LIN {X 0,Y 101.433,Z 824.046,A -85,B 0,C 180,E1 -28794.73,E2 -28794.73} C_VEL
LIN {X 0,Y 101.287,Z 822.969,A -85,B 0,C 180,E1 -28797.017,E2 -28797.017} C_VEL
LIN {X 0,Y 101.21,Z 822.785,A -85,B 0,C 180,E1 -28800.994,E2 -28800.994} C_VEL
LIN {X 0,Y 101.343,Z 823.216,A -85,B 0,C 180,E1 -28803.478,E2 -28803.478} C_VEL
LIN {X 0,Y 102.456,Z 826.592,A -85,B 0,C 180,E1 -28810.373,E2 -28810.373} C_VEL
LIN {X 0,Y 103.056,Z 827.637,A -85,B 0,C 180,E1 -28812.367,E2 -28812.367} C_VEL
LIN {X 0,Y 104.99,Z 831.596,A -85,B 0,C 180,E1 -28817.358,E2 -28817.358} C_VEL
LIN {X 0,Y 106.785,Z 835.312,A -85,B 0,C 180,E1 -28820.877,E2 -28820.877} C_VEL
LIN {X 0,Y 109.032,Z 840.682,A -85,B 0,C 180,E1 -28824.688,E2 -28824.688} C_VEL
LIN {X 0,Y 109.43,Z 842.378,A -85,B 0,C 180,E1 -28825.48,E2 -28825.48} C_VEL
LIN {X 0,Y 107.888,Z 851.485,A -85,B 0,C 180,E1 -28826.117,E2 -28826.117} C_VEL
LIN {X 0,Y 105.588,Z 860.247,A -85,B 0,C 180,E1 -28826.892,E2 -28826.892} C_VEL
LIN {X 0,Y 102.409,Z 869.139,A -85,B 0,C 180,E1 -28827.923,E2 -28827.923} C_VEL
LIN {X 0,Y 98.739,Z 877.424,A -85,B 0,C 180,E1 -28829.317,E2 -28829.317} C_VEL
LIN {X 0,Y 93.703,Z 886.663,A -85,B 0,C 180,E1 -28831.443,E2 -28831.443} C_VEL
LIN {X 0,Y 87.262,Z 896.197,A -85,B 0,C 180,E1 -28834.634,E2 -28834.634} C_VEL
LIN {X 0,Y 82.122,Z 902.568,A -85,B 0,C 180,E1 -28837.663,E2 -28837.663} C_VEL
LIN {X 0,Y 77.037,Z 908.064,A -85,B 0,C 180,E1 -28841.181,E2 -28841.181} C_VEL
LIN {X 0,Y 71.22,Z 913.622,A -85,B 0,C 180,E1 -28846.31,E2 -28846.31} C_VEL
LIN {X 0,Y 65.132,Z 918.794,A -85,B 0,C 180,E1 -28853.596,E2 -28853.596} C_VEL
LIN {X 0,Y 60.395,Z 922.598,A -85,B 0,C 180,E1 -28862.259,E2 -28862.259} C_VEL
LIN {X 0,Y 58.05,Z 924.345,A -85,B 0,C 180,E1 -28868.703,E2 -28868.703} C_VEL
LIN {X 0,Y 56.461,Z 925.598,A -85,B 0,C 180,E1 -28875.585,E2 -28875.585} C_VEL
LIN {X 0,Y 55.612,Z 926.377,A -85,B 0,C 180,E1 -28882.74,E2 -28882.74} C_VEL
LIN {X 0,Y 55.517,Z 926.675,A -85,B 0,C 180,E1 -28890,E2 -28890} C_VEL
LIN {X 0,Y 55.608,Z 926.364,A -85,B 0,C 180,E1 -28897.261,E2 -28897.261} C_VEL
LIN {X 0,Y 56.456,Z 925.559,A -85,B 0,C 180,E1 -28904.417,E2 -28904.417} C_VEL
LIN {X 0,Y 58.05,Z 924.28,A -85,B 0,C 180,E1 -28911.297,E2 -28911.297} C_VEL
LIN {X 0,Y 61.83,Z 921.345,A -85,B 0,C 180,E1 -28920.764,E2 -28920.764} C_VEL
LIN {X 0,Y 65.131,Z 918.672,A -85,B 0,C 180,E1 -28926.404,E2 -28926.404} C_VEL
LIN {X 0,Y 71.219,Z 913.465,A -85,B 0,C 180,E1 -28933.691,E2 -28933.691} C_VEL
LIN {X 0,Y 78.247,Z 906.598,A -85,B 0,C 180,E1 -28939.769,E2 -28939.769} C_VEL
LIN {X 0,Y 84.745,Z 899.107,A -85,B 0,C 180,E1 -28943.958,E2 -28943.958} C_VEL
LIN {X 0,Y 90.162,Z 891.744,A -85,B 0,C 180,E1 -28946.898,E2 -28946.898} C_VEL
LIN {X 0,Y 95.147,Z 883.805,A -85,B 0,C 180,E1 -28949.168,E2 -28949.168} C_VEL
LIN {X 0,Y 100.175,Z 873.929,A -85,B 0,C 180,E1 -28951.279,E2 -28951.279} C_VEL
LIN {X 0,Y 104.464,Z 863.001,A -85,B 0,C 180,E1 -28952.767,E2 -28952.767} C_VEL
LIN {X 0,Y 107.227,Z 853.306,A -85,B 0,C 180,E1 -28953.673,E2 -28953.673} C_VEL
LIN {X 0,Y 109.052,Z 843.744,A -85,B 0,C 180,E1 -28954.304,E2 -28954.304} C_VEL
LIN {X 0,Y 109.146,Z 841.961,A -85,B 0,C 180,E1 -28954.566,E2 -28954.566} C_VEL
LIN {X 0,Y 108.33,Z 839.135,A -85,B 0,C 180,E1 -28956.079,E2 -28956.079} C_VEL
LIN {X 0,Y 105.726,Z 833.29,A -85,B 0,C 180,E1 -28960.588,E2 -28960.588} C_VEL
LIN {X 0,Y 103.976,Z 829.899,A -85,B 0,C 180,E1 -28964.314,E2 -28964.314} C_VEL
LIN {X 0,Y 102.466,Z 826.786,A -85,B 0,C 180,E1 -28968.628,E2 -28968.628} C_VEL
LIN {X 0,Y 101.185,Z 823.736,A -85,B 0,C 180,E1 -28974.895,E2 -28974.895} C_VEL
LIN {X 0,Y 101.064,Z 822.89,A -85,B 0,C 180,E1 -28976.512,E2 -28976.512} C_VEL
LIN {X 0,Y 100.897,Z 822.52,A -85,B 0,C 180,E1 -28980,E2 -28980} C_VEL
LIN {X 0,Y 101.083,Z 823.015,A -85,B 0,C 180,E1 -28984.237,E2 -28984.237} C_VEL
LIN {X 0,Y 102.141,Z 826.386,A -85,B 0,C 180,E1 -28990.756,E2 -28990.756} C_VEL
LIN {X 0,Y 102.807,Z 827.447,A -85,B 0,C 180,E1 -28992.931,E2 -28992.931} C_VEL
LIN {X 0,Y 104.673,Z 831.354,A -85,B 0,C 180,E1 -28997.76,E2 -28997.76} C_VEL
LIN {X 0,Y 106.815,Z 835.705,A -85,B 0,C 180,E1 -29001.883,E2 -29001.883} C_VEL
LIN {X 0,Y 109.044,Z 841.442,A -85,B 0,C 180,E1 -29005.832,E2 -29005.832} C_VEL
LIN {X 0,Y 109.164,Z 841.916,A -85,B 0,C 180,E1 -29006.061,E2 -29006.061} C_VEL
LIN {X 0,Y 107.54,Z 850.651,A -85,B 0,C 180,E1 -29006.759,E2 -29006.759} C_VEL
LIN {X 0,Y 104.166,Z 862.393,A -85,B 0,C 180,E1 -29007.992,E2 -29007.992} C_VEL
LIN {X 0,Y 101.208,Z 869.895,A -85,B 0,C 180,E1 -29009.082,E2 -29009.082} C_VEL
LIN {X 0,Y 98.629,Z 875.115,A -85,B 0,C 180,E1 -29009.687,E2 -29009.687} C_VEL
LIN {X 0,Y 92.879,Z 883.181,A -85,B 0,C 180,E1 -29010.091,E2 -29010.091} C_VEL
LIN {X 0,Y 86.414,Z 890.632,A -85,B 0,C 180,E1 -29010.873,E2 -29010.873} C_VEL
LIN {X 0,Y 82.756,Z 894.84,A -85,B 0,C 180,E1 -29012.187,E2 -29012.187} C_VEL
LIN {X 0,Y 77.419,Z 900.935,A -85,B 0,C 180,E1 -29015.213,E2 -29015.213} C_VEL
LIN {X 0,Y 72.112,Z 906.196,A -85,B 0,C 180,E1 -29018.769,E2 -29018.769} C_VEL
LIN {X 0,Y 67.188,Z 910.582,A -85,B 0,C 180,E1 -29022.928,E2 -29022.928} C_VEL
LIN {X 0,Y 60.547,Z 915.741,A -85,B 0,C 180,E1 -29030.326,E2 -29030.326} C_VEL
LIN {X 0,Y 56.773,Z 918.381,A -85,B 0,C 180,E1 -29036.147,E2 -29036.147} C_VEL
LIN {X 0,Y 52.267,Z 921.272,A -85,B 0,C 180,E1 -29046.21,E2 -29046.21} C_VEL
LIN {X 0,Y 50.185,Z 922.527,A -85,B 0,C 180,E1 -29053.735,E2 -29053.735} C_VEL
LIN {X 0,Y 48.957,Z 923.314,A -85,B 0,C 180,E1 -29061.746,E2 -29061.746} C_VEL
LIN {X 0,Y 48.583,Z 923.612,A -85,B 0,C 180,E1 -29070,E2 -29070} C_VEL
LIN {X 0,Y 48.949,Z 923.331,A -85,B 0,C 180,E1 -29078.255,E2 -29078.255} C_VEL
LIN {X 0,Y 50.169,Z 922.578,A -85,B 0,C 180,E1 -29086.271,E2 -29086.271} C_VEL
LIN {X 0,Y 52.254,Z 921.357,A -85,B 0,C 180,E1 -29093.796,E2 -29093.796} C_VEL
LIN {X 0,Y 56.727,Z 918.502,A -85,B 0,C 180,E1 -29103.884,E2 -29103.884} C_VEL
LIN {X 0,Y 60.499,Z 915.899,A -85,B 0,C 180,E1 -29109.711,E2 -29109.711} C_VEL
LIN {X 0,Y 67.158,Z 910.782,A -85,B 0,C 180,E1 -29117.1,E2 -29117.1} C_VEL
LIN {X 0,Y 73.424,Z 905.271,A -85,B 0,C 180,E1 -29122.155,E2 -29122.155} C_VEL
LIN {X 0,Y 80.103,Z 898.338,A -85,B 0,C 180,E1 -29126.46,E2 -29126.46} C_VEL
LIN {X 0,Y 86.43,Z 890.376,A -85,B 0,C 180,E1 -29129.764,E2 -29129.764} C_VEL
LIN {X 0,Y 91.551,Z 882.781,A -85,B 0,C 180,E1 -29131.983,E2 -29131.983} C_VEL
LIN {X 0,Y 96.169,Z 874.415,A -85,B 0,C 180,E1 -29133.853,E2 -29133.853} C_VEL
LIN {X 0,Y 99.9,Z 866.191,A -85,B 0,C 180,E1 -29135.167,E2 -29135.167} C_VEL
LIN {X 0,Y 103.098,Z 857.074,A -85,B 0,C 180,E1 -29136.303,E2 -29136.303} C_VEL
LIN {X 0,Y 105.754,Z 846.607,A -85,B 0,C 180,E1 -29137.225,E2 -29137.225} C_VEL
LIN {X 0,Y 105.97,Z 845.262,A -85,B 0,C 180,E1 -29137.428,E2 -29137.428} C_VEL
LIN {X 0,Y 104.011,Z 839.684,A -85,B 0,C 180,E1 -29141.924,E2 -29141.924} C_VEL
LIN {X 0,Y 102.747,Z 836.61,A -85,B 0,C 180,E1 -29145.352,E2 -29145.352} C_VEL
LIN {X 0,Y 101.584,Z 833.836,A -85,B 0,C 180,E1 -29149.158,E2 -29149.158} C_VEL
LIN {X 0,Y 100.439,Z 830.717,A -85,B 0,C 180,E1 -29155.987,E2 -29155.987} C_VEL
LIN {X 0,Y 100.366,Z 829.899,A -85,B 0,C 180,E1 -29157.993,E2 -29157.993} C_VEL
LIN {X 0,Y 100.388,Z 829.905,A -85,B 0,C 180,E1 -29162.006,E2 -29162.006} C_VEL
LIN {X 0,Y 101.811,Z 834.378,A -85,B 0,C 180,E1 -29171.32,E2 -29171.32} C_VEL
LIN {X 0,Y 103.551,Z 838.412,A -85,B 0,C 180,E1 -29176.353,E2 -29176.353} C_VEL
LIN {X 0,Y 105.18,Z 842.595,A -85,B 0,C 180,E1 -29180.217,E2 -29180.217} C_VEL
LIN {X 0,Y 106.112,Z 845.288,A -85,B 0,C 180,E1 -29182.18,E2 -29182.18} C_VEL
LIN {X 0,Y 104.361,Z 853.761,A -85,B 0,C 180,E1 -29182.782,E2 -29182.782} C_VEL
LIN {X 0,Y 100.633,Z 865.699,A -85,B 0,C 180,E1 -29183.901,E2 -29183.901} C_VEL
LIN {X 0,Y 96.218,Z 875.717,A -85,B 0,C 180,E1 -29185.324,E2 -29185.324} C_VEL
LIN {X 0,Y 91.688,Z 883.995,A -85,B 0,C 180,E1 -29186.992,E2 -29186.992} C_VEL
LIN {X 0,Y 86.93,Z 891.239,A -85,B 0,C 180,E1 -29188.955,E2 -29188.955} C_VEL
LIN {X 0,Y 82.185,Z 897.466,A -85,B 0,C 180,E1 -29191.224,E2 -29191.224} C_VEL
LIN {X 0,Y 76.601,Z 903.784,A -85,B 0,C 180,E1 -29194.337,E2 -29194.337} C_VEL
LIN {X 0,Y 71.248,Z 909.033,A -85,B 0,C 180,E1 -29197.895,E2 -29197.895} C_VEL
LIN {X 0,Y 66.27,Z 913.414,A -85,B 0,C 180,E1 -29202.067,E2 -29202.067} C_VEL
LIN {X 0,Y 59.544,Z 918.585,A -85,B 0,C 180,E1 -29209.521,E2 -29209.521} C_VEL
LIN {X 0,Y 54.208,Z 922.39,A -85,B 0,C 180,E1 -29218.762,E2 -29218.762} C_VEL
LIN {X 0,Y 51.484,Z 924.137,A -85,B 0,C 180,E1 -29225.825,E2 -29225.825} C_VEL
LIN {X 0,Y 49.598,Z 925.389,A -85,B 0,C 180,E1 -29233.537,E2 -29233.537} C_VEL
LIN {X 0,Y 48.583,Z 926.169,A -85,B 0,C 180,E1 -29241.682,E2 -29241.682} C_VEL
LIN {X 0,Y 48.435,Z 926.467,A -85,B 0,C 180,E1 -29250,E2 -29250} C_VEL
LIN {X 0,Y 48.58,Z 926.155,A -85,B 0,C 180,E1 -29258.318,E2 -29258.318} C_VEL
LIN {X 0,Y 49.593,Z 925.349,A -85,B 0,C 180,E1 -29266.465,E2 -29266.465} C_VEL
LIN {X 0,Y 51.484,Z 924.07,A -85,B 0,C 180,E1 -29274.175,E2 -29274.175} C_VEL
LIN {X 0,Y 55.818,Z 921.134,A -85,B 0,C 180,E1 -29284.513,E2 -29284.513} C_VEL
LIN {X 0,Y 59.543,Z 918.461,A -85,B 0,C 180,E1 -29290.48,E2 -29290.48} C_VEL
LIN {X 0,Y 66.268,Z 913.254,A -85,B 0,C 180,E1 -29297.934,E2 -29297.934} C_VEL
LIN {X 0,Y 73.859,Z 906.386,A -85,B 0,C 180,E1 -29303.98,E2 -29303.98} C_VEL
LIN {X 0,Y 80.77,Z 898.896,A -85,B 0,C 180,E1 -29308.035,E2 -29308.035} C_VEL
LIN {X 0,Y 86.027,Z 892.165,A -85,B 0,C 180,E1 -29310.649,E2 -29310.649} C_VEL
LIN {X 0,Y 90.966,Z 884.824,A -85,B 0,C 180,E1 -29312.683,E2 -29312.683} C_VEL
LIN {X 0,Y 95.443,Z 876.721,A -85,B 0,C 180,E1 -29314.427,E2 -29314.427} C_VEL
LIN {X 0,Y 99.28,Z 868.315,A -85,B 0,C 180,E1 -29315.703,E2 -29315.703} C_VEL
LIN {X 0,Y 102.705,Z 858.796,A -85,B 0,C 180,E1 -29316.704,E2 -29316.704} C_VEL
LIN {X 0,Y 105.706,Z 846.675,A -85,B 0,C 180,E1 -29317.6,E2 -29317.6} C_VEL
LIN {X 0,Y 105.842,Z 844.96,A -85,B 0,C 180,E1 -29317.838,E2 -29317.838} C_VEL
LIN {X 0,Y 103.883,Z 839.468,A -85,B 0,C 180,E1 -29322.197,E2 -29322.197} C_VEL
LIN {X 0,Y 102.288,Z 836.011,A -85,B 0,C 180,E1 -29326.207,E2 -29326.207} C_VEL
LIN {X 0,Y 101.233,Z 833.518,A -85,B 0,C 180,E1 -29329.753,E2 -29329.753} C_VEL
LIN {X 0,Y 100.167,Z 830.206,A -85,B 0,C 180,E1 -29336.481,E2 -29336.481} C_VEL
LIN {X 0,Y 100.04,Z 829.682,A -85,B 0,C 180,E1 -29338.994,E2 -29338.994} C_VEL
LIN {X 0,Y 100.142,Z 830.012,A -85,B 0,C 180,E1 -29343.521,E2 -29343.521} C_VEL
LIN {X 0,Y 101.189,Z 833.514,A -85,B 0,C 180,E1 -29350.568,E2 -29350.568} C_VEL
LIN {X 0,Y 101.932,Z 835.274,A -85,B 0,C 180,E1 -29353.202,E2 -29353.202} C_VEL
LIN {X 0,Y 103.097,Z 837.938,A -85,B 0,C 180,E1 -29356.523,E2 -29356.523} C_VEL
LIN {X 0,Y 104.782,Z 842.217,A -85,B 0,C 180,E1 -29360.612,E2 -29360.612} C_VEL
LIN {X 0,Y 105.791,Z 845.164,A -85,B 0,C 180,E1 -29362.813,E2 -29362.813} C_VEL
LIN {X 0,Y 103.302,Z 855.621,A -85,B 0,C 180,E1 -29363.72,E2 -29363.72} C_VEL
LIN {X 0,Y 99.848,Z 865.466,A -85,B 0,C 180,E1 -29364.789,E2 -29364.789} C_VEL
LIN {X 0,Y 96.407,Z 873.324,A -85,B 0,C 180,E1 -29366.054,E2 -29366.054} C_VEL
LIN {X 0,Y 92.338,Z 881.053,A -85,B 0,C 180,E1 -29367.773,E2 -29367.773} C_VEL
LIN {X 0,Y 87.907,Z 887.928,A -85,B 0,C 180,E1 -29369.607,E2 -29369.607} C_VEL
LIN {X 0,Y 82.756,Z 894.84,A -85,B 0,C 180,E1 -29372.187,E2 -29372.187} C_VEL
LIN {X 0,Y 80.089,Z 897.672,A -85,B 0,C 180,E1 -29373.028,E2 -29373.028} C_VEL
LIN {X 0,Y 74.718,Z 901.732,A -85,B 0,C 180,E1 -29373.377,E2 -29373.377} C_VEL
LIN {X 0,Y 69.197,Z 905.621,A -85,B 0,C 180,E1 -29373.927,E2 -29373.927} C_VEL
LIN {X 0,Y 66.307,Z 907.78,A -85,B 0,C 180,E1 -29375.238,E2 -29375.238} C_VEL
LIN {X 0,Y 60.046,Z 912.696,A -85,B 0,C 180,E1 -29380.466,E2 -29380.466} C_VEL
LIN {X 0,Y 53.082,Z 917.426,A -85,B 0,C 180,E1 -29388.547,E2 -29388.547} C_VEL
LIN {X 0,Y 49.153,Z 919.734,A -85,B 0,C 180,E1 -29395.115,E2 -29395.115} C_VEL
LIN {X 0,Y 45.877,Z 921.481,A -85,B 0,C 180,E1 -29402.64,E2 -29402.64} C_VEL
LIN {X 0,Y 43.42,Z 922.736,A -85,B 0,C 180,E1 -29411.112,E2 -29411.112} C_VEL
LIN {X 0,Y 41.945,Z 923.523,A -85,B 0,C 180,E1 -29420.354,E2 -29420.354} C_VEL
LIN {X 0,Y 41.51,Z 923.82,A -85,B 0,C 180,E1 -29430,E2 -29430} C_VEL
LIN {X 0,Y 41.938,Z 923.539,A -85,B 0,C 180,E1 -29439.647,E2 -29439.647} C_VEL
LIN {X 0,Y 43.407,Z 922.786,A -85,B 0,C 180,E1 -29448.894,E2 -29448.894} C_VEL
LIN {X 0,Y 45.864,Z 921.564,A -85,B 0,C 180,E1 -29457.368,E2 -29457.368} C_VEL
LIN {X 0,Y 50.987,Z 918.71,A -85,B 0,C 180,E1 -29468.337,E2 -29468.337} C_VEL
LIN {X 0,Y 55.223,Z 916.107,A -85,B 0,C 180,E1 -29474.424,E2 -29474.424} C_VEL
LIN {X 0,Y 62.541,Z 910.989,A -85,B 0,C 180,E1 -29481.871,E2 -29481.871} C_VEL
LIN {X 0,Y 69.29,Z 905.479,A -85,B 0,C 180,E1 -29486.803,E2 -29486.803} C_VEL
LIN {X 0,Y 76.419,Z 898.543,A -85,B 0,C 180,E1 -29490.889,E2 -29490.889} C_VEL
LIN {X 0,Y 83.092,Z 890.581,A -85,B 0,C 180,E1 -29493.984,E2 -29493.984} C_VEL
LIN {X 0,Y 88.446,Z 882.985,A -85,B 0,C 180,E1 -29496.037,E2 -29496.037} C_VEL
LIN {X 0,Y 92.76,Z 875.587,A -85,B 0,C 180,E1 -29497.598,E2 -29497.598} C_VEL
LIN {X 0,Y 96.234,Z 868.516,A -85,B 0,C 180,E1 -29498.71,E2 -29498.71} C_VEL
LIN {X 0,Y 99.516,Z 860.219,A -85,B 0,C 180,E1 -29499.698,E2 -29499.698} C_VEL
LIN {X 0,Y 102.34,Z 850.532,A -85,B 0,C 180,E1 -29500.589,E2 -29500.589} C_VEL
LIN {X 0,Y 102.673,Z 848.901,A -85,B 0,C 180,E1 -29500.789,E2 -29500.789} C_VEL
LIN {X 0,Y 101.571,Z 844.575,A -85,B 0,C 180,E1 -29504.922,E2 -29504.922} C_VEL
LIN {X 0,Y 100.264,Z 840.614,A -85,B 0,C 180,E1 -29510.162,E2 -29510.162} C_VEL
LIN {X 0,Y 99.495,Z 837.257,A -85,B 0,C 180,E1 -29517.469,E2 -29517.469} C_VEL
LIN {X 0,Y 99.474,Z 836.759,A -85,B 0,C 180,E1 -29520,E2 -29520} C_VEL
LIN {X 0,Y 99.499,Z 837.152,A -85,B 0,C 180,E1 -29522.023,E2 -29522.023} C_VEL
LIN {X 0,Y 100.476,Z 841.22,A -85,B 0,C 180,E1 -29530.325,E2 -29530.325} C_VEL
LIN {X 0,Y 101.8,Z 845.01,A -85,B 0,C 180,E1 -29535.184,E2 -29535.184} C_VEL
LIN {X 0,Y 102.936,Z 848.909,A -85,B 0,C 180,E1 -29538.794,E2 -29538.794} C_VEL
LIN {X 0,Y 100.36,Z 858.656,A -85,B 0,C 180,E1 -29539.503,E2 -29539.503} C_VEL
LIN {X 0,Y 97.391,Z 866.859,A -85,B 0,C 180,E1 -29540.263,E2 -29540.263} C_VEL
LIN {X 0,Y 93.402,Z 875.513,A -85,B 0,C 180,E1 -29541.384,E2 -29541.384} C_VEL
LIN {X 0,Y 88.686,Z 883.789,A -85,B 0,C 180,E1 -29542.892,E2 -29542.892} C_VEL
LIN {X 0,Y 83.396,Z 891.461,A -85,B 0,C 180,E1 -29544.814,E2 -29544.814} C_VEL
LIN {X 0,Y 78.732,Z 897.26,A -85,B 0,C 180,E1 -29546.792,E2 -29546.792} C_VEL
LIN {X 0,Y 72.837,Z 903.578,A -85,B 0,C 180,E1 -29549.726,E2 -29549.726} C_VEL
LIN {X 0,Y 67.11,Z 908.826,A -85,B 0,C 180,E1 -29553.092,E2 -29553.092} C_VEL
LIN {X 0,Y 61.743,Z 913.207,A -85,B 0,C 180,E1 -29557.175,E2 -29557.175} C_VEL
LIN {X 0,Y 54.324,Z 918.377,A -85,B 0,C 180,E1 -29564.639,E2 -29564.639} C_VEL
LIN {X 0,Y 48.258,Z 922.182,A -85,B 0,C 180,E1 -29574.371,E2 -29574.371} C_VEL
LIN {X 0,Y 45.094,Z 923.928,A -85,B 0,C 180,E1 -29582.124,E2 -29582.124} C_VEL
LIN {X 0,Y 42.829,Z 925.181,A -85,B 0,C 180,E1 -29590.841,E2 -29590.841} C_VEL
LIN {X 0,Y 41.564,Z 925.96,A -85,B 0,C 180,E1 -29600.265,E2 -29600.265} C_VEL
LIN {X 0,Y 41.337,Z 926.258,A -85,B 0,C 180,E1 -29610,E2 -29610} C_VEL
LIN {X 0,Y 41.562,Z 925.946,A -85,B 0,C 180,E1 -29619.735,E2 -29619.735} C_VEL
LIN {X 0,Y 42.825,Z 925.14,A -85,B 0,C 180,E1 -29629.161,E2 -29629.161} C_VEL
LIN {X 0,Y 45.094,Z 923.86,A -85,B 0,C 180,E1 -29637.876,E2 -29637.876} C_VEL
LIN {X 0,Y 50.108,Z 920.923,A -85,B 0,C 180,E1 -29649.135,E2 -29649.135} C_VEL
LIN {X 0,Y 54.324,Z 918.25,A -85,B 0,C 180,E1 -29655.361,E2 -29655.361} C_VEL
LIN {X 0,Y 61.741,Z 913.044,A -85,B 0,C 180,E1 -29662.827,E2 -29662.827} C_VEL
LIN {X 0,Y 69.921,Z 906.175,A -85,B 0,C 180,E1 -29668.689,E2 -29668.689} C_VEL
LIN {X 0,Y 77.245,Z 898.684,A -85,B 0,C 180,E1 -29672.51,E2 -29672.51} C_VEL
LIN {X 0,Y 83.423,Z 891.121,A -85,B 0,C 180,E1 -29675.153,E2 -29675.153} C_VEL
LIN {X 0,Y 88.705,Z 883.378,A -85,B 0,C 180,E1 -29677.078,E2 -29677.078} C_VEL
LIN {X 0,Y 94.187,Z 873.502,A -85,B 0,C 180,E1 -29678.863,E2 -29678.863} C_VEL
LIN {X 0,Y 98.777,Z 862.568,A -85,B 0,C 180,E1 -29680.111,E2 -29680.111} C_VEL
LIN {X 0,Y 101.806,Z 852.559,A -85,B 0,C 180,E1 -29680.875,E2 -29680.875} C_VEL
LIN {X 0,Y 102.706,Z 848.701,A -85,B 0,C 180,E1 -29681.162,E2 -29681.162} C_VEL
LIN {X 0,Y 101.438,Z 844.506,A -85,B 0,C 180,E1 -29685.096,E2 -29685.096} C_VEL
LIN {X 0,Y 100.396,Z 841.59,A -85,B 0,C 180,E1 -29688.798,E2 -29688.798} C_VEL
LIN {X 0,Y 99.977,Z 840.259,A -85,B 0,C 180,E1 -29690.798,E2 -29690.798} C_VEL
LIN {X 0,Y 99.213,Z 836.86,A -85,B 0,C 180,E1 -29697.971,E2 -29697.971} C_VEL
LIN {X 0,Y 99.192,Z 836.804,A -85,B 0,C 180,E1 -29702.031,E2 -29702.031} C_VEL
LIN {X 0,Y 100.167,Z 841.039,A -85,B 0,C 180,E1 -29710.869,E2 -29710.869} C_VEL
LIN {X 0,Y 101.431,Z 844.812,A -85,B 0,C 180,E1 -29715.632,E2 -29715.632} C_VEL
LIN {X 0,Y 102.468,Z 848.815,A -85,B 0,C 180,E1 -29719.443,E2 -29719.443} C_VEL
LIN {X 0,Y 100.206,Z 857.211,A -85,B 0,C 180,E1 -29720.145,E2 -29720.145} C_VEL
LIN {X 0,Y 97.048,Z 865.779,A -85,B 0,C 180,E1 -29721.001,E2 -29721.001} C_VEL
LIN {X 0,Y 93.513,Z 873.538,A -85,B 0,C 180,E1 -29722.153,E2 -29722.153} C_VEL
LIN {X 0,Y 89.255,Z 881.266,A -85,B 0,C 180,E1 -29723.742,E2 -29723.742} C_VEL
LIN {X 0,Y 84.632,Z 888.14,A -85,B 0,C 180,E1 -29725.435,E2 -29725.435} C_VEL
LIN {X 0,Y 79.026,Z 895.259,A -85,B 0,C 180,E1 -29727.927,E2 -29727.927} C_VEL
LIN {X 0,Y 73.553,Z 901.147,A -85,B 0,C 180,E1 -29730.689,E2 -29730.689} C_VEL
LIN {X 0,Y 67.9,Z 906.406,A -85,B 0,C 180,E1 -29734.102,E2 -29734.102} C_VEL
LIN {X 0,Y 66.307,Z 907.78,A -85,B 0,C 180,E1 -29735.238,E2 -29735.238} C_VEL
LIN {X 0,Y 62.183,Z 910.911,A -85,B 0,C 180,E1 -29737.787,E2 -29737.787} C_VEL
LIN {X 0,Y 54.178,Z 915.363,A -85,B 0,C 180,E1 -29741.55,E2 -29741.55} C_VEL
LIN {X 0,Y 46.12,Z 918.874,A -85,B 0,C 180,E1 -29746.882,E2 -29746.882} C_VEL
LIN {X 0,Y 42.19,Z 920.509,A -85,B 0,C 180,E1 -29752.234,E2 -29752.234} C_VEL
LIN {X 0,Y 36.792,Z 922.945,A -85,B 0,C 180,E1 -29767.54,E2 -29767.54} C_VEL
LIN {X 0,Y 34.982,Z 923.731,A -85,B 0,C 180,E1 -29778.41,E2 -29778.41} C_VEL
LIN {X 0,Y 34.422,Z 924.029,A -85,B 0,C 180,E1 -29790,E2 -29790} C_VEL
LIN {X 0,Y 34.977,Z 923.748,A -85,B 0,C 180,E1 -29801.591,E2 -29801.591} C_VEL
LIN {X 0,Y 36.781,Z 922.994,A -85,B 0,C 180,E1 -29812.467,E2 -29812.467} C_VEL
LIN {X 0,Y 39.692,Z 921.773,A -85,B 0,C 180,E1 -29822.086,E2 -29822.086} C_VEL
LIN {X 0,Y 45.623,Z 918.918,A -85,B 0,C 180,E1 -29833.884,E2 -29833.884} C_VEL
LIN {X 0,Y 50.403,Z 916.314,A -85,B 0,C 180,E1 -29840.076,E2 -29840.076} C_VEL
LIN {X 0,Y 58.425,Z 911.197,A -85,B 0,C 180,E1 -29847.355,E2 -29847.355} C_VEL
LIN {X 0,Y 65.666,Z 905.686,A -85,B 0,C 180,E1 -29852.002,E2 -29852.002} C_VEL
LIN {X 0,Y 73.231,Z 898.749,A -85,B 0,C 180,E1 -29855.744,E2 -29855.744} C_VEL
LIN {X 0,Y 80.235,Z 890.786,A -85,B 0,C 180,E1 -29858.54,E2 -29858.54} C_VEL
LIN {X 0,Y 85.81,Z 883.19,A -85,B 0,C 180,E1 -29860.368,E2 -29860.368} C_VEL
LIN {X 0,Y 90.8,Z 874.858,A -85,B 0,C 180,E1 -29861.899,E2 -29861.899} C_VEL
LIN {X 0,Y 94.687,Z 866.9,A -85,B 0,C 180,E1 -29862.94,E2 -29862.94} C_VEL
LIN {X 0,Y 98.305,Z 857.352,A -85,B 0,C 180,E1 -29863.9,E2 -29863.9} C_VEL
LIN {X 0,Y 99.359,Z 854.143,A -85,B 0,C 180,E1 -29864.171,E2 -29864.171} C_VEL
LIN {X 0,Y 99.618,Z 852.251,A -85,B 0,C 180,E1 -29864.787,E2 -29864.787} C_VEL
LIN {X 0,Y 98.966,Z 849.128,A -85,B 0,C 180,E1 -29868.56,E2 -29868.56} C_VEL
LIN {X 0,Y 98.557,Z 846.956,A -85,B 0,C 180,E1 -29872.088,E2 -29872.088} C_VEL
LIN {X 0,Y 98.322,Z 843.888,A -85,B 0,C 180,E1 -29878.976,E2 -29878.976} C_VEL
LIN {X 0,Y 98.324,Z 843.997,A -85,B 0,C 180,E1 -29881.151,E2 -29881.151} C_VEL
LIN {X 0,Y 98.838,Z 847.695,A -85,B 0,C 180,E1 -29888.94,E2 -29888.94} C_VEL
LIN {X 0,Y 99.584,Z 851.198,A -85,B 0,C 180,E1 -29893.65,E2 -29893.65} C_VEL
LIN {X 0,Y 99.852,Z 852.893,A -85,B 0,C 180,E1 -29895.233,E2 -29895.233} C_VEL
LIN {X 0,Y 96.161,Z 864.326,A -85,B 0,C 180,E1 -29896.003,E2 -29896.003} C_VEL
LIN {X 0,Y 91.871,Z 873.806,A -85,B 0,C 180,E1 -29897.014,E2 -29897.014} C_VEL
LIN {X 0,Y 86.98,Z 882.353,A -85,B 0,C 180,E1 -29898.304,E2 -29898.304} C_VEL
LIN {X 0,Y 81.201,Z 890.588,A -85,B 0,C 180,E1 -29900.069,E2 -29900.069} C_VEL
LIN {X 0,Y 75.792,Z 897.053,A -85,B 0,C 180,E1 -29901.986,E2 -29901.986} C_VEL
LIN {X 0,Y 69.584,Z 903.371,A -85,B 0,C 180,E1 -29904.632,E2 -29904.632} C_VEL
LIN {X 0,Y 63.506,Z 908.618,A -85,B 0,C 180,E1 -29907.707,E2 -29907.707} C_VEL
LIN {X 0,Y 57.727,Z 912.999,A -85,B 0,C 180,E1 -29911.546,E2 -29911.546} C_VEL
LIN {X 0,Y 49.586,Z 918.169,A -85,B 0,C 180,E1 -29918.782,E2 -29918.782} C_VEL
LIN {X 0,Y 42.675,Z 921.973,A -85,B 0,C 180,E1 -29928.795,E2 -29928.795} C_VEL
LIN {X 0,Y 38.959,Z 923.72,A -85,B 0,C 180,E1 -29937.236,E2 -29937.236} C_VEL
LIN {X 0,Y 36.199,Z 924.972,A -85,B 0,C 180,E1 -29947.151,E2 -29947.151} C_VEL
LIN {X 0,Y 34.575,Z 925.751,A -85,B 0,C 180,E1 -29958.272,E2 -29958.272} C_VEL
LIN {X 0,Y 34.253,Z 926.05,A -85,B 0,C 180,E1 -29970,E2 -29970} C_VEL
LIN {X 0,Y 34.573,Z 925.737,A -85,B 0,C 180,E1 -29981.729,E2 -29981.729} C_VEL
LIN {X 0,Y 36.196,Z 924.931,A -85,B 0,C 180,E1 -29992.85,E2 -29992.85} C_VEL
LIN {X 0,Y 38.959,Z 923.65,A -85,B 0,C 180,E1 -30002.764,E2 -30002.764} C_VEL
LIN {X 0,Y 44.795,Z 920.712,A -85,B 0,C 180,E1 -30014.911,E2 -30014.911} C_VEL
LIN {X 0,Y 49.585,Z 918.04,A -85,B 0,C 180,E1 -30021.219,E2 -30021.219} C_VEL
LIN {X 0,Y 57.725,Z 912.833,A -85,B 0,C 180,E1 -30028.456,E2 -30028.456} C_VEL
LIN {X 0,Y 66.512,Z 905.965,A -85,B 0,C 180,E1 -30033.916,E2 -30033.916} C_VEL
LIN {X 0,Y 74.226,Z 898.472,A -85,B 0,C 180,E1 -30037.394,E2 -30037.394} C_VEL
LIN {X 0,Y 80.248,Z 891.474,A -85,B 0,C 180,E1 -30039.599,E2 -30039.599} C_VEL
LIN {X 0,Y 85.384,Z 884.398,A -85,B 0,C 180,E1 -30041.186,E2 -30041.186} C_VEL
LIN {X 0,Y 90.228,Z 876.294,A -85,B 0,C 180,E1 -30042.587,E2 -30042.587} C_VEL
LIN {X 0,Y 94.338,Z 867.886,A -85,B 0,C 180,E1 -30043.569,E2 -30043.569} C_VEL
LIN {X 0,Y 97.965,Z 858.363,A -85,B 0,C 180,E1 -30044.349,E2 -30044.349} C_VEL
LIN {X 0,Y 99.662,Z 852.435,A -85,B 0,C 180,E1 -30044.769,E2 -30044.769} C_VEL
LIN {X 0,Y 98.886,Z 848.954,A -85,B 0,C 180,E1 -30048.859,E2 -30048.859} C_VEL
LIN {X 0,Y 98.411,Z 846.813,A -85,B 0,C 180,E1 -30052.305,E2 -30052.305} C_VEL
LIN {X 0,Y 98.037,Z 843.756,A -85,B 0,C 180,E1 -30058.974,E2 -30058.974} C_VEL
LIN {X 0,Y 98.021,Z 843.966,A -85,B 0,C 180,E1 -30062.055,E2 -30062.055} C_VEL
LIN {X 0,Y 98.48,Z 847.685,A -85,B 0,C 180,E1 -30069.719,E2 -30069.719} C_VEL
LIN {X 0,Y 99.151,Z 851.078,A -85,B 0,C 180,E1 -30074.236,E2 -30074.236} C_VEL
LIN {X 0,Y 99.466,Z 852.578,A -85,B 0,C 180,E1 -30075.842,E2 -30075.842} C_VEL
LIN {X 0,Y 95.465,Z 864.369,A -85,B 0,C 180,E1 -30076.854,E2 -30076.854} C_VEL
LIN {X 0,Y 90.921,Z 874.04,A -85,B 0,C 180,E1 -30078.062,E2 -30078.062} C_VEL
LIN {X 0,Y 86.645,Z 881.478,A -85,B 0,C 180,E1 -30079.45,E2 -30079.45} C_VEL
LIN {X 0,Y 81.839,Z 888.351,A -85,B 0,C 180,E1 -30080.949,E2 -30080.949} C_VEL
LIN {X 0,Y 76.37,Z 895.029,A -85,B 0,C 180,E1 -30083.036,E2 -30083.036} C_VEL
LIN {X 0,Y 70.199,Z 901.358,A -85,B 0,C 180,E1 -30085.705,E2 -30085.705} C_VEL
LIN {X 0,Y 64.198,Z 906.616,A -85,B 0,C 180,E1 -30088.861,E2 -30088.861} C_VEL
LIN {X 0,Y 58.45,Z 911.003,A -85,B 0,C 180,E1 -30092.682,E2 -30092.682} C_VEL
LIN {X 0,Y 50.447,Z 916.161,A -85,B 0,C 180,E1 -30099.983,E2 -30099.983} C_VEL
LIN {X 0,Y 45.683,Z 918.801,A -85,B 0,C 180,E1 -30106.188,E2 -30106.188} C_VEL
LIN {X 0,Y 42.19,Z 920.509,A -85,B 0,C 180,E1 -30112.234,E2 -30112.234} C_VEL
LIN {X 0,Y 38.661,Z 921.957,A -85,B 0,C 180,E1 -30118.695,E2 -30118.695} C_VEL
LIN {X 0,Y 34.851,Z 923.026,A -85,B 0,C 180,E1 -30125.634,E2 -30125.634} C_VEL
LIN {X 0,Y 28.546,Z 924.09,A -85,B 0,C 180,E1 -30144.048,E2 -30144.048} C_VEL
LIN {X 0,Y 27.502,Z 924.147,A -85,B 0,C 180,E1 -30156.05,E2 -30156.05} C_VEL
LIN {X 0,Y 27.662,Z 924.042,A -85,B 0,C 180,E1 -30160.155,E2 -30160.155} C_VEL
LIN {X 0,Y 30.348,Z 923.202,A -85,B 0,C 180,E1 -30177.592,E2 -30177.592} C_VEL
LIN {X 0,Y 33.894,Z 921.981,A -85,B 0,C 180,E1 -30188.467,E2 -30188.467} C_VEL
LIN {X 0,Y 40.798,Z 919.126,A -85,B 0,C 180,E1 -30200.822,E2 -30200.822} C_VEL
LIN {X 0,Y 46.165,Z 916.522,A -85,B 0,C 180,E1 -30206.857,E2 -30206.857} C_VEL
LIN {X 0,Y 54.922,Z 911.404,A -85,B 0,C 180,E1 -30213.603,E2 -30213.603} C_VEL
LIN {X 0,Y 62.647,Z 905.893,A -85,B 0,C 180,E1 -30217.748,E2 -30217.748} C_VEL
LIN {X 0,Y 70.611,Z 898.956,A -85,B 0,C 180,E1 -30221.004,E2 -30221.004} C_VEL
LIN {X 0,Y 77.921,Z 890.992,A -85,B 0,C 180,E1 -30223.398,E2 -30223.398} C_VEL
LIN {X 0,Y 83.696,Z 883.394,A -85,B 0,C 180,E1 -30224.942,E2 -30224.942} C_VEL
LIN {X 0,Y 88.038,Z 876.529,A -85,B 0,C 180,E1 -30226.062,E2 -30226.062} C_VEL
LIN {X 0,Y 92.586,Z 867.705,A -85,B 0,C 180,E1 -30227.066,E2 -30227.066} C_VEL
LIN {X 0,Y 95.876,Z 859.583,A -85,B 0,C 180,E1 -30227.802,E2 -30227.802} C_VEL
LIN {X 0,Y 96.296,Z 858.372,A -85,B 0,C 180,E1 -30227.887,E2 -30227.887} C_VEL
LIN {X 0,Y 96.815,Z 856.431,A -85,B 0,C 180,E1 -30228.482,E2 -30228.482} C_VEL
LIN {X 0,Y 96.627,Z 853.714,A -85,B 0,C 180,E1 -30232.687,E2 -30232.687} C_VEL
LIN {X 0,Y 96.732,Z 850.689,A -85,B 0,C 180,E1 -30240,E2 -30240} C_VEL
LIN {X 0,Y 96.809,Z 854.417,A -85,B 0,C 180,E1 -30248.085,E2 -30248.085} C_VEL
LIN {X 0,Y 97.049,Z 856.376,A -85,B 0,C 180,E1 -30250.975,E2 -30250.975} C_VEL
LIN {X 0,Y 96.585,Z 858.159,A -85,B 0,C 180,E1 -30251.531,E2 -30251.531} C_VEL
LIN {X 0,Y 92.964,Z 867.476,A -85,B 0,C 180,E1 -30252.14,E2 -30252.14} C_VEL
LIN {X 0,Y 89.191,Z 875.14,A -85,B 0,C 180,E1 -30252.869,E2 -30252.869} C_VEL
LIN {X 0,Y 84.177,Z 883.378,A -85,B 0,C 180,E1 -30253.932,E2 -30253.932} C_VEL
LIN {X 0,Y 78.367,Z 891.221,A -85,B 0,C 180,E1 -30255.411,E2 -30255.411} C_VEL
LIN {X 0,Y 71.796,Z 898.555,A -85,B 0,C 180,E1 -30257.367,E2 -30257.367} C_VEL
LIN {X 0,Y 63.719,Z 905.998,A -85,B 0,C 180,E1 -30260.36,E2 -30260.36} C_VEL
LIN {X 0,Y 55.885,Z 911.832,A -85,B 0,C 180,E1 -30264.252,E2 -30264.252} C_VEL
LIN {X 0,Y 48.347,Z 916.435,A -85,B 0,C 180,E1 -30269.285,E2 -30269.285} C_VEL
LIN {X 0,Y 42.685,Z 919.43,A -85,B 0,C 180,E1 -30274.589,E2 -30274.589} C_VEL
LIN {X 0,Y 37.598,Z 921.764,A -85,B 0,C 180,E1 -30281.608,E2 -30281.608} C_VEL
LIN {X 0,Y 33.189,Z 923.511,A -85,B 0,C 180,E1 -30290.559,E2 -30290.559} C_VEL
LIN {X 0,Y 29.765,Z 924.763,A -85,B 0,C 180,E1 -30301.821,E2 -30301.821} C_VEL
LIN {X 0,Y 27.663,Z 925.542,A -85,B 0,C 180,E1 -30315.282,E2 -30315.282} C_VEL
LIN {X 0,Y 27.145,Z 925.841,A -85,B 0,C 180,E1 -30330,E2 -30330} C_VEL
LIN {X 0,Y 27.661,Z 925.528,A -85,B 0,C 180,E1 -30344.719,E2 -30344.719} C_VEL
LIN {X 0,Y 29.763,Z 924.721,A -85,B 0,C 180,E1 -30358.182,E2 -30358.182} C_VEL
LIN {X 0,Y 33.189,Z 923.44,A -85,B 0,C 180,E1 -30369.441,E2 -30369.441} C_VEL
LIN {X 0,Y 40.062,Z 920.501,A -85,B 0,C 180,E1 -30382.132,E2 -30382.132} C_VEL
LIN {X 0,Y 45.471,Z 917.829,A -85,B 0,C 180,E1 -30388.22,E2 -30388.22} C_VEL
LIN {X 0,Y 54.342,Z 912.622,A -85,B 0,C 180,E1 -30394.865,E2 -30394.865} C_VEL
LIN {X 0,Y 63.714,Z 905.754,A -85,B 0,C 180,E1 -30399.651,E2 -30399.651} C_VEL
LIN {X 0,Y 71.79,Z 898.259,A -85,B 0,C 180,E1 -30402.649,E2 -30402.649} C_VEL
LIN {X 0,Y 78.215,Z 891.075,A -85,B 0,C 180,E1 -30404.513,E2 -30404.513} C_VEL
LIN {X 0,Y 83.363,Z 884.185,A -85,B 0,C 180,E1 -30405.818,E2 -30405.818} C_VEL
LIN {X 0,Y 88.285,Z 876.219,A -85,B 0,C 180,E1 -30406.97,E2 -30406.97} C_VEL
LIN {X 0,Y 92.264,Z 868.378,A -85,B 0,C 180,E1 -30407.726,E2 -30407.726} C_VEL
LIN {X 0,Y 95.549,Z 860.281,A -85,B 0,C 180,E1 -30408.285,E2 -30408.285} C_VEL
LIN {X 0,Y 96.499,Z 857.558,A -85,B 0,C 180,E1 -30408.452,E2 -30408.452} C_VEL
LIN {X 0,Y 96.829,Z 856.128,A -85,B 0,C 180,E1 -30409.008,E2 -30409.008} C_VEL
LIN {X 0,Y 96.428,Z 853.33,A -85,B 0,C 180,E1 -30413.461,E2 -30413.461} C_VEL
LIN {X 0,Y 96.434,Z 850.633,A -85,B 0,C 180,E1 -30419.479,E2 -30419.479} C_VEL
LIN {X 0,Y 96.352,Z 850.96,A -85,B 0,C 180,E1 -30421.568,E2 -30421.568} C_VEL
LIN {X 0,Y 96.416,Z 854.086,A -85,B 0,C 180,E1 -30428.383,E2 -30428.383} C_VEL
LIN {X 0,Y 96.556,Z 856.508,A -85,B 0,C 180,E1 -30431.863,E2 -30431.863} C_VEL
LIN {X 0,Y 96.025,Z 858.29,A -85,B 0,C 180,E1 -30432.246,E2 -30432.246} C_VEL
LIN {X 0,Y 93.16,Z 865.671,A -85,B 0,C 180,E1 -30432.776,E2 -30432.776} C_VEL
LIN {X 0,Y 89.052,Z 874.117,A -85,B 0,C 180,E1 -30433.696,E2 -30433.696} C_VEL
LIN {X 0,Y 84.549,Z 881.691,A -85,B 0,C 180,E1 -30434.914,E2 -30434.914} C_VEL
LIN {X 0,Y 79.58,Z 888.563,A -85,B 0,C 180,E1 -30436.177,E2 -30436.177} C_VEL
LIN {X 0,Y 73.887,Z 895.24,A -85,B 0,C 180,E1 -30437.976,E2 -30437.976} C_VEL
LIN {X 0,Y 67.429,Z 901.568,A -85,B 0,C 180,E1 -30440.273,E2 -30440.273} C_VEL
LIN {X 0,Y 61.096,Z 906.827,A -85,B 0,C 180,E1 -30443.036,E2 -30443.036} C_VEL
LIN {X 0,Y 54.943,Z 911.213,A -85,B 0,C 180,E1 -30446.44,E2 -30446.44} C_VEL
LIN {X 0,Y 46.209,Z 916.371,A -85,B 0,C 180,E1 -30453.228,E2 -30453.228} C_VEL
LIN {X 0,Y 40.85,Z 919.011,A -85,B 0,C 180,E1 -30459.267,E2 -30459.267} C_VEL
LIN {X 0,Y 33.907,Z 921.9,A -85,B 0,C 180,E1 -30471.55,E2 -30471.55} C_VEL
LIN {X 0,Y 30.356,Z 923.154,A -85,B 0,C 180,E1 -30482.417,E2 -30482.417} C_VEL
LIN {X 0,Y 28.074,Z 923.94,A -85,B 0,C 180,E1 -30495.503,E2 -30495.503} C_VEL
LIN {X 0,Y 27.349,Z 924.237,A -85,B 0,C 180,E1 -30510,E2 -30510} C_VEL
LIN {X 0,Y 27.662,Z 924.042,A -85,B 0,C 180,E1 -30520.155,E2 -30520.155} C_VEL
LIN {X 0,Y 28.457,Z 923.689,A -85,B 0,C 180,E1 -30532.081,E2 -30532.081} C_VEL
LIN {X 0,Y 30.447,Z 922.35,A -85,B 0,C 180,E1 -30550.877,E2 -30550.877} C_VEL
LIN {X 0,Y 34.955,Z 920.198,A -85,B 0,C 180,E1 -30566.043,E2 -30566.043} C_VEL
LIN {X 0,Y 39.186,Z 918.368,A -85,B 0,C 180,E1 -30571.916,E2 -30571.916} C_VEL
LIN {X 0,Y 48.963,Z 913.513,A -85,B 0,C 180,E1 -30578.907,E2 -30578.907} C_VEL
LIN {X 0,Y 57.029,Z 908.437,A -85,B 0,C 180,E1 -30582.76,E2 -30582.76} C_VEL
LIN {X 0,Y 63.63,Z 903.47,A -85,B 0,C 180,E1 -30585.116,E2 -30585.116} C_VEL
LIN {X 0,Y 70.312,Z 897.475,A -85,B 0,C 180,E1 -30587.049,E2 -30587.049} C_VEL
LIN {X 0,Y 77.033,Z 890.181,A -85,B 0,C 180,E1 -30588.744,E2 -30588.744} C_VEL
LIN {X 0,Y 82.883,Z 882.523,A -85,B 0,C 180,E1 -30589.881,E2 -30589.881} C_VEL
LIN {X 0,Y 88.105,Z 874.098,A -85,B 0,C 180,E1 -30590.882,E2 -30590.882} C_VEL
LIN {X 0,Y 92.96,Z 864.197,A -85,B 0,C 180,E1 -30591.672,E2 -30591.672} C_VEL
LIN {X 0,Y 93.562,Z 862.8,A -85,B 0,C 180,E1 -30591.759,E2 -30591.759} C_VEL
LIN {X 0,Y 94.114,Z 860.981,A -85,B 0,C 180,E1 -30592.382,E2 -30592.382} C_VEL
LIN {X 0,Y 94.172,Z 860.222,A -85,B 0,C 180,E1 -30593.57,E2 -30593.57} C_VEL
LIN {X 0,Y 94.596,Z 857.721,A -85,B 0,C 180,E1 -30600,E2 -30600} C_VEL
LIN {X 0,Y 94.287,Z 860.815,A -85,B 0,C 180,E1 -30606.974,E2 -30606.974} C_VEL
LIN {X 0,Y 93.945,Z 862.102,A -85,B 0,C 180,E1 -30607.545,E2 -30607.545} C_VEL
LIN {X 0,Y 89.06,Z 872.877,A -85,B 0,C 180,E1 -30608.176,E2 -30608.176} C_VEL
LIN {X 0,Y 83.615,Z 881.943,A -85,B 0,C 180,E1 -30609.028,E2 -30609.028} C_VEL
LIN {X 0,Y 77.553,Z 890.093,A -85,B 0,C 180,E1 -30610.138,E2 -30610.138} C_VEL
LIN {X 0,Y 71.689,Z 896.64,A -85,B 0,C 180,E1 -30611.379,E2 -30611.379} C_VEL
LIN {X 0,Y 64.958,Z 902.957,A -85,B 0,C 180,E1 -30613.16,E2 -30613.16} C_VEL
LIN {X 0,Y 58.273,Z 908.204,A -85,B 0,C 180,E1 -30615.24,E2 -30615.24} C_VEL
LIN {X 0,Y 51.722,Z 912.584,A -85,B 0,C 180,E1 -30617.981,E2 -30617.981} C_VEL
LIN {X 0,Y 42.164,Z 917.753,A -85,B 0,C 180,E1 -30623.543,E2 -30623.543} C_VEL
LIN {X 0,Y 33.288,Z 921.555,A -85,B 0,C 180,E1 -30632.38,E2 -30632.38} C_VEL
LIN {X 0,Y 28.051,Z 923.302,A -85,B 0,C 180,E1 -30641.267,E2 -30641.267} C_VEL
LIN {X 0,Y 23.735,Z 924.554,A -85,B 0,C 180,E1 -30653.686,E2 -30653.686} C_VEL
LIN {X 0,Y 20.884,Z 925.333,A -85,B 0,C 180,E1 -30670.335,E2 -30670.335} C_VEL
LIN {X 0,Y 20.039,Z 925.631,A -85,B 0,C 180,E1 -30690,E2 -30690} C_VEL
LIN {X 0,Y 20.882,Z 925.319,A -85,B 0,C 180,E1 -30709.667,E2 -30709.667} C_VEL
LIN {X 0,Y 23.733,Z 924.511,A -85,B 0,C 180,E1 -30726.317,E2 -30726.317} C_VEL
LIN {X 0,Y 28.05,Z 923.23,A -85,B 0,C 180,E1 -30738.733,E2 -30738.733} C_VEL
LIN {X 0,Y 36.129,Z 920.291,A -85,B 0,C 180,E1 -30751.087,E2 -30751.087} C_VEL
LIN {X 0,Y 42.163,Z 917.619,A -85,B 0,C 180,E1 -30756.458,E2 -30756.458} C_VEL
LIN {X 0,Y 51.721,Z 912.411,A -85,B 0,C 180,E1 -30762.023,E2 -30762.023} C_VEL
LIN {X 0,Y 61.609,Z 905.543,A -85,B 0,C 180,E1 -30765.842,E2 -30765.842} C_VEL
LIN {X 0,Y 70.029,Z 898.015,A -85,B 0,C 180,E1 -30768.228,E2 -30768.228} C_VEL
LIN {X 0,Y 76.629,Z 890.863,A -85,B 0,C 180,E1 -30769.624,E2 -30769.624} C_VEL
LIN {X 0,Y 81.909,Z 883.972,A -85,B 0,C 180,E1 -30770.654,E2 -30770.654} C_VEL
LIN {X 0,Y 86.744,Z 876.384,A -85,B 0,C 180,E1 -30771.497,E2 -30771.497} C_VEL
LIN {X 0,Y 91.329,Z 867.491,A -85,B 0,C 180,E1 -30772.134,E2 -30772.134} C_VEL
LIN {X 0,Y 93.694,Z 861.939,A -85,B 0,C 180,E1 -30772.43,E2 -30772.43} C_VEL
LIN {X 0,Y 94.065,Z 860.571,A -85,B 0,C 180,E1 -30773.003,E2 -30773.003} C_VEL
LIN {X 0,Y 94.385,Z 857.411,A -85,B 0,C 180,E1 -30780,E2 -30780} C_VEL
LIN {X 0,Y 93.884,Z 860.704,A -85,B 0,C 180,E1 -30787.637,E2 -30787.637} C_VEL
LIN {X 0,Y 93.873,Z 860.892,A -85,B 0,C 180,E1 -30787.919,E2 -30787.919} C_VEL
LIN {X 0,Y 92.357,Z 864.798,A -85,B 0,C 180,E1 -30788.407,E2 -30788.407} C_VEL
LIN {X 0,Y 88.256,Z 873.257,A -85,B 0,C 180,E1 -30789.077,E2 -30789.077} C_VEL
LIN {X 0,Y 83.008,Z 881.903,A -85,B 0,C 180,E1 -30790.183,E2 -30790.183} C_VEL
LIN {X 0,Y 77.903,Z 888.775,A -85,B 0,C 180,E1 -30791.162,E2 -30791.162} C_VEL
LIN {X 0,Y 72.018,Z 895.451,A -85,B 0,C 180,E1 -30792.611,E2 -30792.611} C_VEL
LIN {X 0,Y 65.314,Z 901.779,A -85,B 0,C 180,E1 -30794.436,E2 -30794.436} C_VEL
LIN {X 0,Y 58.689,Z 907.037,A -85,B 0,C 180,E1 -30796.664,E2 -30796.664} C_VEL
LIN {X 0,Y 52.171,Z 911.424,A -85,B 0,C 180,E1 -30799.444,E2 -30799.444} C_VEL
LIN {X 0,Y 42.73,Z 916.582,A -85,B 0,C 180,E1 -30805.229,E2 -30805.229} C_VEL
LIN {X 0,Y 36.766,Z 919.221,A -85,B 0,C 180,E1 -30810.66,E2 -30810.66} C_VEL
LIN {X 0,Y 28.684,Z 922.109,A -85,B 0,C 180,E1 -30822.689,E2 -30822.689} C_VEL
LIN {X 0,Y 24.284,Z 923.364,A -85,B 0,C 180,E1 -30834.633,E2 -30834.633} C_VEL
LIN {X 0,Y 21.274,Z 924.149,A -85,B 0,C 180,E1 -30850.71,E2 -30850.71} C_VEL
LIN {X 0,Y 20.257,Z 924.446,A -85,B 0,C 180,E1 -30870,E2 -30870} C_VEL
LIN {X 0,Y 21.27,Z 924.165,A -85,B 0,C 180,E1 -30889.294,E2 -30889.294} C_VEL
LIN {X 0,Y 24.277,Z 923.411,A -85,B 0,C 180,E1 -30905.379,E2 -30905.379} C_VEL
LIN {X 0,Y 28.672,Z 922.189,A -85,B 0,C 180,E1 -30917.337,E2 -30917.337} C_VEL
LIN {X 0,Y 36.725,Z 919.334,A -85,B 0,C 180,E1 -30929.447,E2 -30929.447} C_VEL
LIN {X 0,Y 39.186,Z 918.368,A -85,B 0,C 180,E1 -30931.916,E2 -30931.916} C_VEL
LIN {X 0,Y 43.648,Z 916.376,A -85,B 0,C 180,E1 -30936.552,E2 -30936.552} C_VEL
LIN {X 0,Y 50.4,Z 912.433,A -85,B 0,C 180,E1 -30944.052,E2 -30944.052} C_VEL
LIN {X 0,Y 57.306,Z 907.537,A -85,B 0,C 180,E1 -30949.597,E2 -30949.597} C_VEL
LIN {X 0,Y 61.734,Z 904.048,A -85,B 0,C 180,E1 -30951.336,E2 -30951.336} C_VEL
LIN {X 0,Y 69.071,Z 897.681,A -85,B 0,C 180,E1 -30952.781,E2 -30952.781} C_VEL
LIN {X 0,Y 75.968,Z 890.386,A -85,B 0,C 180,E1 -30953.994,E2 -30953.994} C_VEL
LIN {X 0,Y 80.791,Z 884.346,A -85,B 0,C 180,E1 -30954.606,E2 -30954.606} C_VEL
LIN {X 0,Y 85.716,Z 876.968,A -85,B 0,C 180,E1 -30955.296,E2 -30955.296} C_VEL
LIN {X 0,Y 90.617,Z 867.803,A -85,B 0,C 180,E1 -30955.864,E2 -30955.864} C_VEL
LIN {X 0,Y 91.454,Z 865.926,A -85,B 0,C 180,E1 -30956.384,E2 -30956.384} C_VEL
LIN {X 0,Y 91.979,Z 864.584,A -85,B 0,C 180,E1 -30960,E2 -30960} C_VEL
LIN {X 0,Y 91.518,Z 866.047,A -85,B 0,C 180,E1 -30963.321,E2 -30963.321} C_VEL
LIN {X 0,Y 86.823,Z 875.268,A -85,B 0,C 180,E1 -30963.748,E2 -30963.748} C_VEL
LIN {X 0,Y 81.926,Z 882.969,A -85,B 0,C 180,E1 -30964.25,E2 -30964.25} C_VEL
LIN {X 0,Y 75.84,Z 890.808,A -85,B 0,C 180,E1 -30965.003,E2 -30965.003} C_VEL
LIN {X 0,Y 68.09,Z 898.94,A -85,B 0,C 180,E1 -30966.123,E2 -30966.123} C_VEL
LIN {X 0,Y 58.545,Z 906.821,A -85,B 0,C 180,E1 -30967.958,E2 -30967.958} C_VEL
LIN {X 0,Y 49.985,Z 912.376,A -85,B 0,C 180,E1 -30970.193,E2 -30970.193} C_VEL
LIN {X 0,Y 39.862,Z 917.545,A -85,B 0,C 180,E1 -30974.14,E2 -30974.14} C_VEL
LIN {X 0,Y 30.076,Z 921.346,A -85,B 0,C 180,E1 -30980.822,E2 -30980.822} C_VEL
LIN {X 0,Y 23.959,Z 923.093,A -85,B 0,C 180,E1 -30988.355,E2 -30988.355} C_VEL
LIN {X 0,Y 18.495,Z 924.345,A -85,B 0,C 180,E1 -31000.536,E2 -31000.536} C_VEL
LIN {X 0,Y 14.391,Z 925.124,A -85,B 0,C 180,E1 -31020.766,E2 -31020.766} C_VEL
LIN {X 0,Y 12.948,Z 925.423,A -85,B 0,C 180,E1 -31050,E2 -31050} C_VEL
LIN {X 0,Y 14.389,Z 925.11,A -85,B 0,C 180,E1 -31079.237,E2 -31079.237} C_VEL
LIN {X 0,Y 18.494,Z 924.302,A -85,B 0,C 180,E1 -31099.467,E2 -31099.467} C_VEL
LIN {X 0,Y 23.959,Z 923.019,A -85,B 0,C 180,E1 -31111.645,E2 -31111.645} C_VEL
LIN {X 0,Y 33.277,Z 920.081,A -85,B 0,C 180,E1 -31121.875,E2 -31121.875} C_VEL
LIN {X 0,Y 39.862,Z 917.409,A -85,B 0,C 180,E1 -31125.86,E2 -31125.86} C_VEL
LIN {X 0,Y 49.984,Z 912.2,A -85,B 0,C 180,E1 -31129.812,E2 -31129.812} C_VEL
LIN {X 0,Y 58.543,Z 906.604,A -85,B 0,C 180,E1 -31132.054,E2 -31132.054} C_VEL
LIN {X 0,Y 67.918,Z 898.801,A -85,B 0,C 180,E1 -31133.862,E2 -31133.862} C_VEL
LIN {X 0,Y 74.975,Z 891.469,A -85,B 0,C 180,E1 -31134.853,E2 -31134.853} C_VEL
LIN {X 0,Y 81.06,Z 883.759,A -85,B 0,C 180,E1 -31135.611,E2 -31135.611} C_VEL
LIN {X 0,Y 85.617,Z 876.799,A -85,B 0,C 180,E1 -31136.142,E2 -31136.142} C_VEL
LIN {X 0,Y 89.954,Z 868.725,A -85,B 0,C 180,E1 -31136.544,E2 -31136.544} C_VEL
LIN {X 0,Y 90.63,Z 867.276,A -85,B 0,C 180,E1 -31136.588,E2 -31136.588} C_VEL
LIN {X 0,Y 91.441,Z 865.32,A -85,B 0,C 180,E1 -31137.648,E2 -31137.648} C_VEL
LIN {X 0,Y 91.787,Z 864.306,A -85,B 0,C 180,E1 -31140,E2 -31140} C_VEL
LIN {X 0,Y 91.216,Z 865.779,A -85,B 0,C 180,E1 -31143.868,E2 -31143.868} C_VEL
LIN {X 0,Y 88.853,Z 870.88,A -85,B 0,C 180,E1 -31144.318,E2 -31144.318} C_VEL
LIN {X 0,Y 82.818,Z 881.031,A -85,B 0,C 180,E1 -31145.195,E2 -31145.195} C_VEL
LIN {X 0,Y 76.845,Z 888.987,A -85,B 0,C 180,E1 -31145.96,E2 -31145.96} C_VEL
LIN {X 0,Y 70.808,Z 895.663,A -85,B 0,C 180,E1 -31147,E2 -31147} C_VEL
LIN {X 0,Y 63.918,Z 901.99,A -85,B 0,C 180,E1 -31148.279,E2 -31148.279} C_VEL
LIN {X 0,Y 57.063,Z 907.247,A -85,B 0,C 180,E1 -31149.834,E2 -31149.834} C_VEL
LIN {X 0,Y 50.256,Z 911.634,A -85,B 0,C 180,E1 -31151.789,E2 -31151.789} C_VEL
LIN {X 0,Y 40.22,Z 916.792,A -85,B 0,C 180,E1 -31156.039,E2 -31156.039} C_VEL
LIN {X 0,Y 33.703,Z 919.43,A -85,B 0,C 180,E1 -31160.218,E2 -31160.218} C_VEL
LIN {X 0,Y 24.436,Z 922.319,A -85,B 0,C 180,E1 -31170.364,E2 -31170.364} C_VEL
LIN {X 0,Y 18.951,Z 923.573,A -85,B 0,C 180,E1 -31182.124,E2 -31182.124} C_VEL
LIN {X 0,Y 14.766,Z 924.358,A -85,B 0,C 180,E1 -31201.578,E2 -31201.578} C_VEL
LIN {X 0,Y 13.179,Z 924.654,A -85,B 0,C 180,E1 -31230,E2 -31230} C_VEL
LIN {X 0,Y 14.762,Z 924.373,A -85,B 0,C 180,E1 -31258.43,E2 -31258.43} C_VEL
LIN {X 0,Y 18.946,Z 923.619,A -85,B 0,C 180,E1 -31277.893,E2 -31277.893} C_VEL
LIN {X 0,Y 24.427,Z 922.397,A -85,B 0,C 180,E1 -31289.671,E2 -31289.671} C_VEL
LIN {X 0,Y 33.676,Z 919.542,A -85,B 0,C 180,E1 -31299.906,E2 -31299.906} C_VEL
LIN {X 0,Y 40.202,Z 916.937,A -85,B 0,C 180,E1 -31304.05,E2 -31304.05} C_VEL
LIN {X 0,Y 50.246,Z 911.819,A -85,B 0,C 180,E1 -31308.269,E2 -31308.269} C_VEL
LIN {X 0,Y 58.761,Z 906.307,A -85,B 0,C 180,E1 -31310.656,E2 -31310.656} C_VEL
LIN {X 0,Y 61.734,Z 904.048,A -85,B 0,C 180,E1 -31311.336,E2 -31311.336} C_VEL
LIN {X 0,Y 64.596,Z 901.661,A -85,B 0,C 180,E1 -31312.545,E2 -31312.545} C_VEL
LIN {X 0,Y 68.751,Z 897.757,A -85,B 0,C 180,E1 -31315.69,E2 -31315.69} C_VEL
LIN {X 0,Y 72.85,Z 893.679,A -85,B 0,C 180,E1 -31318.515,E2 -31318.515} C_VEL
LIN {X 0,Y 75.402,Z 890.77,A -85,B 0,C 180,E1 -31319.333,E2 -31319.333} C_VEL
LIN {X 0,Y 77.311,Z 888.556,A -85,B 0,C 180,E1 -31319.525,E2 -31319.525} C_VEL
LIN {X 0,Y 70.28,Z 896.227,A -85,B 0,C 180,E1 -31319.934,E2 -31319.934} C_VEL
LIN {X 0,Y 63.255,Z 902.543,A -85,B 0,C 180,E1 -31320.513,E2 -31320.513} C_VEL
LIN {X 0,Y 56.235,Z 907.79,A -85,B 0,C 180,E1 -31321.152,E2 -31321.152} C_VEL
LIN {X 0,Y 49.226,Z 912.167,A -85,B 0,C 180,E1 -31321.999,E2 -31321.999} C_VEL
LIN {X 0,Y 38.744,Z 917.338,A -85,B 0,C 180,E1 -31323.905,E2 -31323.905} C_VEL
LIN {X 0,Y 28.336,Z 921.137,A -85,B 0,C 180,E1 -31327.215,E2 -31327.215} C_VEL
LIN {X 0,Y 21.511,Z 922.884,A -85,B 0,C 180,E1 -31331.43,E2 -31331.43} C_VEL
LIN {X 0,Y 14.883,Z 924.136,A -85,B 0,C 180,E1 -31339.193,E2 -31339.193} C_VEL
LIN {X 0,Y 8.9,Z 924.916,A -85,B 0,C 180,E1 -31357.848,E2 -31357.848} C_VEL
LIN {X 0,Y 5.868,Z 925.214,A -85,B 0,C 180,E1 -31410,E2 -31410} C_VEL
LIN {X 0,Y 8.899,Z 924.901,A -85,B 0,C 180,E1 -31462.158,E2 -31462.158} C_VEL
LIN {X 0,Y 14.883,Z 924.092,A -85,B 0,C 180,E1 -31480.812,E2 -31480.812} C_VEL
LIN {X 0,Y 21.511,Z 922.809,A -85,B 0,C 180,E1 -31488.57,E2 -31488.57} C_VEL
LIN {X 0,Y 31.792,Z 919.871,A -85,B 0,C 180,E1 -31494.144,E2 -31494.144} C_VEL
LIN {X 0,Y 38.744,Z 917.199,A -85,B 0,C 180,E1 -31496.096,E2 -31496.096} C_VEL
LIN {X 0,Y 49.226,Z 911.989,A -85,B 0,C 180,E1 -31498.008,E2 -31498.008} C_VEL
LIN {X 0,Y 59.744,Z 905.121,A -85,B 0,C 180,E1 -31499.175,E2 -31499.175} C_VEL
LIN {X 0,Y 67.529,Z 898.589,A -85,B 0,C 180,E1 -31499.88,E2 -31499.88} C_VEL
LIN {X 0,Y 74.674,Z 891.256,A -85,B 0,C 180,E1 -31500.289,E2 -31500.289} C_VEL
LIN {X 0,Y 77.31,Z 888.188,A -85,B 0,C 180,E1 -31500.421,E2 -31500.421} C_VEL
LIN {X 0,Y 77.312,Z 888.181,A -85,B 0,C 180,E1 -31500.601,E2 -31500.601} C_VEL
LIN {X 0,Y 70.297,Z 895.874,A -85,B 0,C 180,E1 -31501.245,E2 -31501.245} C_VEL
LIN {X 0,Y 63.288,Z 902.2,A -85,B 0,C 180,E1 -31501.924,E2 -31501.924} C_VEL
LIN {X 0,Y 56.287,Z 907.457,A -85,B 0,C 180,E1 -31502.71,E2 -31502.71} C_VEL
LIN {X 0,Y 49.298,Z 911.845,A -85,B 0,C 180,E1 -31503.686,E2 -31503.686} C_VEL
LIN {X 0,Y 38.862,Z 917.002,A -85,B 0,C 180,E1 -31505.935,E2 -31505.935} C_VEL
LIN {X 0,Y 31.952,Z 919.64,A -85,B 0,C 180,E1 -31508.189,E2 -31508.189} C_VEL
LIN {X 0,Y 21.732,Z 922.528,A -85,B 0,C 180,E1 -31514.021,E2 -31514.021} C_VEL
LIN {X 0,Y 15.141,Z 923.781,A -85,B 0,C 180,E1 -31521.825,E2 -31521.825} C_VEL
LIN {X 0,Y 9.179,Z 924.566,A -85,B 0,C 180,E1 -31540.031,E2 -31540.031} C_VEL
LIN {X 0,Y 6.094,Z 924.862,A -85,B 0,C 180,E1 -31590,E2 -31590} C_VEL
LIN {X 0,Y 9.176,Z 924.582,A -85,B 0,C 180,E1 -31639.985,E2 -31639.985} C_VEL
LIN {X 0,Y 15.139,Z 923.827,A -85,B 0,C 180,E1 -31658.199,E2 -31658.199} C_VEL
LIN {X 0,Y 21.727,Z 922.605,A -85,B 0,C 180,E1 -31666.026,E2 -31666.026} C_VEL
LIN {X 0,Y 31.941,Z 919.75,A -85,B 0,C 180,E1 -31671.943,E2 -31671.943} C_VEL
LIN {X 0,Y 38.856,Z 917.145,A -85,B 0,C 180,E1 -31674.155,E2 -31674.155} C_VEL
LIN {X 0,Y 49.295,Z 912.026,A -85,B 0,C 180,E1 -31676.375,E2 -31676.375} C_VEL
LIN {X 0,Y 58.033,Z 906.513,A -85,B 0,C 180,E1 -31677.572,E2 -31677.572} C_VEL
LIN {X 0,Y 66.789,Z 899.573,A -85,B 0,C 180,E1 -31678.511,E2 -31678.511} C_VEL
LIN {X 0,Y 74.679,Z 891.608,A -85,B 0,C 180,E1 -31679.246,E2 -31679.246} C_VEL
LIN {X 0,Y 75.402,Z 890.77,A -85,B 0,C 180,E1 -31679.333,E2 -31679.333} C_VEL
LIN {X 0,Y 75.402,Z 890.77,A -85,B 0,C 180,E1 -31679.333,E2 -31679.333}

QRS_NEXT_CUT()

QRS_NEXT()
QRS_HOME()

END
